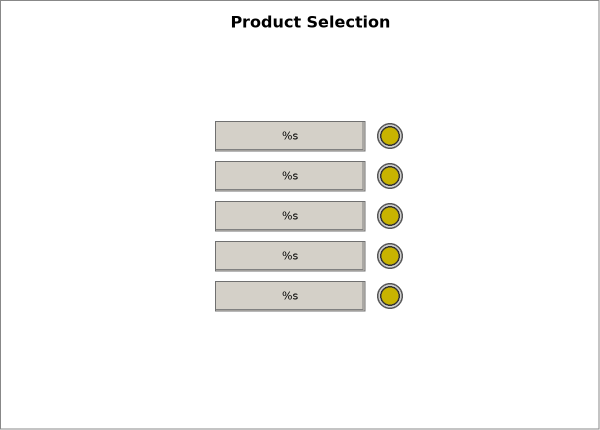
VISUALIZATION Manual_Select_Tube  // 600x430
    Button (215,121 150x30), "%s", text variable: MAIN.TubeSelection[1].ProductName
        OnMouseClick: execute {
            MAIN.TubeHmi := MAIN.TubeSelection[1];
            MAIN.fbSlitter.Manual.bCameraSelectTube := TRUE;
            MAIN.TubeIndicator[1] := TRUE;
            MAIN.TubeIndicator[2] := FALSE;
            MAIN.TubeIndicator[3] := FALSE;
            MAIN.TubeIndicator[4] := FALSE;
            MAIN.TubeIndicator[5] := FALSE;
        }
    Button (215,161 150x30), "%s", text variable: MAIN.TubeSelection[2].ProductName
        OnMouseClick: execute {
            MAIN.TubeHmi := MAIN.TubeSelection[2];
            MAIN.fbSlitter.Manual.bCameraSelectTube := TRUE;
            MAIN.TubeIndicator[1] := FALSE;
            MAIN.TubeIndicator[2] := TRUE;
            MAIN.TubeIndicator[3] := FALSE;
            MAIN.TubeIndicator[4] := FALSE;
            MAIN.TubeIndicator[5] := FALSE;
        }
    Button (215,201 150x30), "%s", text variable: MAIN.TubeSelection[3].ProductName
        OnMouseClick: execute {
            MAIN.TubeHmi := MAIN.TubeSelection[3];
            MAIN.fbSlitter.Manual.bCameraSelectTube := TRUE;
            MAIN.TubeIndicator[1] := FALSE;
            MAIN.TubeIndicator[2] := FALSE;
            MAIN.TubeIndicator[3] := TRUE;
            MAIN.TubeIndicator[4] := FALSE;
            MAIN.TubeIndicator[5] := FALSE;
        }
    Button (215,241 150x30), "%s", text variable: MAIN.TubeSelection[4].ProductName
        OnMouseClick: execute {
            MAIN.TubeHmi := MAIN.TubeSelection[4];
            MAIN.fbSlitter.Manual.bCameraSelectTube := TRUE;
            MAIN.TubeIndicator[1] := FALSE;
            MAIN.TubeIndicator[2] := FALSE;
            MAIN.TubeIndicator[3] := FALSE;
            MAIN.TubeIndicator[4] := TRUE;
            MAIN.TubeIndicator[5] := FALSE;
        }
    Button (215,281 150x30), "%s", text variable: MAIN.TubeSelection[5].ProductName
        OnMouseClick: execute {
            MAIN.TubeHmi := MAIN.TubeSelection[5];
            MAIN.fbSlitter.Manual.bCameraSelectTube := TRUE;
            MAIN.TubeIndicator[1] := FALSE;
            MAIN.TubeIndicator[2] := FALSE;
            MAIN.TubeIndicator[3] := FALSE;
            MAIN.TubeIndicator[4] := FALSE;
            MAIN.TubeIndicator[5] := TRUE;
        }
    Lamp1 (375,121 30x30), variable: MAIN.TubeIndicator[1], style: Lamp-Lamp1-Yellow
    Lamp1 (375,161 30x30), variable: MAIN.TubeIndicator[2], style: Lamp-Lamp1-Yellow
    Lamp1 (375,201 30x30), variable: MAIN.TubeIndicator[3], style: Lamp-Lamp1-Yellow
    Lamp1 (375,241 30x30), variable: MAIN.TubeIndicator[4], style: Lamp-Lamp1-Yellow
    Lamp1 (375,281 30x30), variable: MAIN.TubeIndicator[5], style: Lamp-Lamp1-Yellow
    Label (133,7 355x30), "Product Selection"
END_VISUALIZATION

(* stored: Version 1.1.0.1, ProductVersion 3.1.4024.3
   Visu Manual_Select_Tube: Id {78d7784b-f26f-4f5d-b903-44d0835e388d} *)
